PROGRAM Ax7
VAR
	iAxisNumber : INT := E_AxisNames.Sample_Stack_X_Translation;
	iGroupNumber : INT := 3;
	
	stoRTrig : R_Trig;
END_VAR

//Initial parameters of an Axis
IF _TaskInfo[fbGetCurTaskIndex.index].FirstCycle THEN
    //Initial default values:
    GVL.astAxes[iAxisNumber].stHomingConfig.eHomeSeq :=E_HomingRoutines.eHomeToRef_Bwd;
    GVL.astAxes[iAxisNumber].stHomingConfig.fHomePosition := 0.0;
    GVL.astAxes[iAxisNumber].stHomingConfig.fHomeFinishDistance := 0.0;
    GVL.astAxes[iAxisNumber].stConfig.eRestorePosition := E_RestorePosition.eRestoreWithoutHome;
	GVL.astAxes[iAxisNumber].stControl.bAutoEnableDisable := TRUE;
	GVL.astAxes[iAxisNumber].stControl.tMoveFinishedDelay := T#0.1S;
	//Set which group this axis belongs to
	GVL.astAxes[iAxisNumber].stDescription.iGroupNumber := iGroupNumber;
	GVL.astAxes[iAxisNumber].Commissioning := TRUE;
END_IF

stoRTrig(CLK:=GVL.astAxes[iAxisNumber].stStatus.bSTOActive);
IF stoRTrig.Q THEN
	GVL.astAxes[iAxisNumber].stControl.bReset:= TRUE;
END_IF

IF SAFETY.STOP_MOTION THEN
	GVL.astAxes[iAxisNumber].stControl.bHalt:= TRUE;
END_IF


//Define ACTIONS() or write exclusive code for an specific axis.
(*Eg. Stop when temperature reaches certain values, reduce speed if  a signal is activated, etc.
Eg. GVL.astAxes[x].stControl.bInterlockFwd := NOT bInterlockFwdOK;*)

END_PROGRAM

(* stored: Version 1.1.0.1, ProductVersion 3.1.4026.18
   POU Ax7: Id {46130b17-40a1-4690-bc14-8240edfa58c7}, SpecialFunc None *)
